FUNCTION_BLOCK PushPopFB
VAR_INPUT
	Push:BOOL;
	Pop: BOOL;
	PushNumber: UINT;
END_VAR
VAR_OUTPUT
	TargetFloor: UINT;
END_VAR
VAR
	Queue: ARRAY [1..3] OF UINT:=[0,0,0];
	numberExist : BOOL;
	i: INT:=1;
END_VAR



IF Push THEN
    numberExist := FALSE;
    FOR i:=1 TO 3 DO
        IF Queue[i] = PushNumber THEN
            numberExist := TRUE;
            EXIT; // Exit as soon as a duplicate is found
        END_IF
    END_FOR

    IF NOT numberExist THEN
        FOR i:=1 TO 3 DO
            IF Queue[i] = 0 THEN
                Queue[i] := PushNumber;
                EXIT; // Exit after inserting the number to the first empty slot
            END_IF
        END_FOR
    END_IF
END_IF



IF Pop THEN
	FOR i:=1 TO 2 DO
		Queue[i]:=Queue[i+1];
	END_FOR
	Queue[3]:=0;
END_IF


// Store Target Floor

FOR i:=1 TO 3 DO
	IF Queue[i] <> 0 THEN
		TargetFloor := Queue[i];
		EXIT;
	END_IF
END_FOR

END_FUNCTION_BLOCK

(* stored: Version 1.1.0.1, ProductVersion 3.1.4024.12
   POU PushPopFB: Id {ed9cf65b-112f-43d1-ab41-4e08b8b5abe1}, SpecialFunc None *)
